// TIA Portal V18 export
DATA_BLOCK "Heater settings"   // DB138
{ S7_Optimized_Access := 'TRUE' }
VERSION : 0.1
// stored: AutoNumber true, DBAccessibleFromOPCUA true, IsOnlyStoredInLoadMemory false, IsRetainMemResEnabled false, IsWriteProtectedInAS false, MemoryReserve 100
   VAR RETAIN
      "Heater 1" : Struct
         "set temperature" : Real;
         "preshutdown temperature" : Real;
         "Limit under temparature" : Real;
         "Limit Over temperature" : Real;
         "Heating adjustment hysteresis" : Real;
         "Minimum ON time" : Real;
         "Minimum Off time" : Real;
      END_STRUCT;
      "Heater 2" : Struct
         "set temperature" : Real;
         "preshutdown temperature" : Real;
         "Limit under temparature" : Real;
         "Limit Over temperature" : Real;
         "Heating adjustment hysteresis" : Real;
         "Minimum ON time" : Real;
         "Minimum Off time" : Real;
      END_STRUCT;
      "Heater 3" : Struct
         "set temperature" : Real;
         "preshutdown temperature" : Real;
         "Limit under temparature" : Real;
         "Limit Over temperature" : Real;
         "Heating adjustment hysteresis" : Real;
         "Minimum ON time" : Real;
         "Minimum Off time" : Real;
      END_STRUCT;
      "Heater 4" : Struct
         "set temperature" : Real;
         "preshutdown temperature" : Real;
         "Limit under temparature" : Real;
         "Limit Over temperature" : Real;
         "Heating adjustment hysteresis" : Real;
         "Minimum ON time" : Real;
         "Minimum Off time" : Real;
      END_STRUCT;
      "heater EN 1" : Bool;
      "heater EN 2" : Bool;
      "heater EN 3" : Bool;
      "heater EN 4" : Bool;
   END_VAR
BEGIN
END_DATA_BLOCK
